# B&R Automation Studio project CControl_Gschneitner (part 18)

```automation-basic
		ENDACTION

	ENDCASE

	InitOK = 1

END_PROGRAM
```

#### CSV01_PRGInit.ab
```automation-basic
PROGRAM _INIT

; Diverse INIT :
; ==============
  InitOK = 0
  CSV01.IW.KOPF_WRITE           = 0
  CSV01.IW.DATA_WRITE           = 0
  CSV01.IW.DATA_WRITE_BEREIT    = 0
  CSV01.IW.RPS_SAVE_STEP_Nr     = 0
  CSV01.IW.RPS_CPYDEL_STEP_Nr   = 0
  CSV01.IW.RPS_DirRead_Start_OK = 0

  M_DatObj_ChangDate = DT#1970-01-01-00:00:00

  strcpy(adr(CSV01.IW.PC_Device), "PC_HD_D")		; PC: Speicherdevice
  strcpy(adr(DatObjInfo_01_Name), "CSV01_CFG")

  CR = $0D			; CR (Enter)
  LF = $0A			; LF (Linefeed)
  StrCRLF[0] = CR	; CR+LF
  StrCRLF[1] = LF	; CR+LF
  StrCRLF[2] = 0	; CR+LF
  StrCRLF[3] = 0	; CR+LF

; Task-Zykluszeit auslesen:
; =========================
  RTInfo(1, RT_Status, ZyklTime, init_reason, task_class)
  ZyklTime = ZyklTime/1000  ; [msek]

END_PROGRAM
```

#### CSV01_PRG.var
```iecst
VAR
	CR : USINT;
	CSV_DatObj1 : CSV_DatObj1_typ;
	CSV_DatObj2 : CSV_DatObj2_typ;
	data_len : UDINT;
	data_len2 : UDINT;
	data_typ : UDINT;
	Datei_Ende : ARRAY[0..1] OF USINT;
	Datensatz : ARRAY[0..60000] OF USINT;
	DatObj_Offset : UDINT;
	DatObj1_Size : UDINT;
	DatObj2_Size : UDINT;
	DatObjInfo_01 : DatObjInfo;
	DatObjInfo_01_Name : ARRAY[0..15] OF USINT;
	DevLink_0 : DevLink;
	DevMemInfo_0 : DevMemInfo;
	dimension : UINT;
	DirCopy_0 : DirCopy;
	DirCreate_0 : DirCreate;
	DirDeleteEx_0 : DirDeleteEx;
	DirInfo_0 : DirInfo;
	DirRead_0 : DirRead;
	DirRead_alt_Date : DATE_AND_TIME;
	DirRead_alt_entry : UDINT;
	DirRead_entry : UDINT;
	DirRead_neu_Date : DATE_AND_TIME;
	DirRead_neu_entry : UDINT;
	DirRead_Nr : UDINT;
	ET : UDINT;
	FileClose_0 : FileClose;
	FileCopy_0 : FileCopy;
	FileCreate_0 : FileCreate;
	FileDelete_0 : FileDelete;
	FileIdent : UDINT;
	FileLength : UDINT;
	FileOpen_0 : FileOpen;
	FileRead_0 : FileRead;
	FileWrite_0 : FileWrite;
	i : UINT;
	ii : UINT;
	init_reason : SINT;
	InitOK : BOOL;
	LF : USINT;
	M_date_Fehler : BOOL;
	M_DatObj_ChangDate : DATE_AND_TIME;
	M_Fehler : BOOL;
	M_File_neu : BOOL;
	M_InitOK : BOOL;
	M_MAX_Fehler : BOOL;
	M_MIN_Fehler : BOOL;
	M_Tag_ID : ARRAY[0..9999] OF BOOL;
	M_Tag_MAX : LREAL;
	M_Tag_MIN : LREAL;
	M_timestamp_Fehler : BOOL;
	M_timestamp_QM_Fehler : BOOL;
	M_UDINT_Fehler : BOOL;
	nxt_adr : UDINT;
	Offset_Ende : UDINT;
	P_Fehler : REFERENCE TO BOOL;
	P_Warnung : REFERENCE TO BOOL;
	pv_adr : UDINT;
	RT_Status : UINT;
	RTC_gettime_Status : UINT;
	status_adr : UINT;
	status_ninfo : UINT;
	Str_date : STRING[10];
	Str_ID : ARRAY[0..11] OF USINT;
	Str_Min : ARRAY[0..11] OF USINT;
	Str_Nachkomma : ARRAY[0..11] OF USINT;
	Str_QM_timestamp : STRING[14];
	Str_RPS_File_Name : ARRAY[0..300] OF USINT;
	Str_Sek : ARRAY[0..11] OF USINT;
	Str_Std : ARRAY[0..11] OF USINT;
	Str_Stellen : ARRAY[0..11] OF USINT;
	Str_timestamp : STRING[23];
	Str_Ziel_File_Name : ARRAY[0..300] OF USINT;
	StrCRLF : ARRAY[0..3] OF USINT;
	StrWork : ARRAY[0..30] OF USINT;
	Tag_MAX_Komma : USINT;
	Tag_MAX_Nachkomma : USINT;
	Tag_MAX_Stellen : USINT;
	Tag_MIN_Komma : USINT;
	Tag_MIN_Nachkomma : USINT;
	Tag_MIN_Stellen : USINT;
	Tag_Nachkomma : USINT;
	task_class : SINT;
	Wert_BOOL : REFERENCE TO BOOL;
	Wert_DINT : DINT;
	Wert_INT : INT;
	Wert_REAL : REAL;
	Wert_SINT : SINT;
	Wert_STRING : ARRAY[0..24] OF USINT;
	Wert_UDINT : UDINT;
	Wert_UINT : UINT;
	Wert_USINT : USINT;
	Zeile_Fertig : BOOL;
	ZyklTime : UDINT;
END_VAR
```

### Data object Logical/CSV/CSV01_CFG (Simple, version 1.00.0) - Tag Configuration

#### CSV01_CFG.dat
```
; ============================================================================================
; ACHTUNG: !!! In diesem Datenmodul dürfen absolut keine Tabulator-Sprünge enthalten sein !!!!
; ============================================================================================

;[ABSCHNITT_CONFIG]
;******************

;<----------------->   -> Länge der 8 nachstehenden Eingabefelder
"1.0.0.1            "  ; USINT[0..19] CSV-Version für Auswertung in Reporting-Software                  z.B.: "1.0.0.1            "
"LATronicCControl   "  ; USINT[0..19] Anlagenname                                                       z.B.: "Heizung_01         "
"CF                 "  ; USINT[0..19]          RPS-Ebene: File-Devicename (CPU Eigenschaften)           z.B.: "CF                 "
"CSV                "  ; USINT[0..19]          RPS-Ebene: Zielordner (nur eine Hirachieebene möglich)   z.B.: "CSV                "
"usb_device         "  ; USINT[0..19] [OPTION] EXTERN   : File-Devicename (CPU Eigenschaften)           z.B.: "USB                "
"CSV                "  ; USINT[0..19] [OPTION] EXTERN   : Zielordner (nur eine Hirachieebene möglich)   z.B.: "CSV                "
"192.168.203.202    "  ; USINT[0..19] [OPTION] PC-Ebene : IP-Adresse PC                                 z.B.: "192.168.203.204    "
"PC_D               "  ; USINT[0..19] [OPTION] PC-Ebene : Windows-Freigabename des Laufwerks am PC  	z.B.: "PC_D               "
"guest              "  ; USINT[0..19] [OPTION] PC-Ebene : Windows-Username (nicht akt. Anmeldung verw.) z.B.: "guest              "
"guest              "  ; USINT[0..19] [OPTION] PC-Ebene : Windows-Userpassword                      	z.B.: "guest              "
"/Daten/Excel/CSV                                                                                   " ;USINT[0..99] [OPTION] PC-Ebene: Zielordner (muß am PC manuell angelegt werden
;<------------------------------------------------------------------------------------------------->

;[ABSCHNITT_DATEN]
;*****************

;TAG-ID          TAG-Variablenname (RPS-Name)                                  TAG-Bezeichung                                   TAG-Einheit                  TAG-MIN           TAG-MAX
;[DINT]                USINT[0..47]                                             USINT[0..59]                                    USINT[0..31]                USINT[0..15]      USINT[0..15]
; 0..9999
;(mit "0"          (RPS-Variablenname)                                          (freier Text)                                   (freier Text)               (Komma=".")       (Komma=".")
;auffüllen!)                                                                                                                                               (=Trend SkalaU)    (=Trend SkalaO)
;                                                                                                                                                          (=Def. Kommast.)  (=Def. Kommast.)
;---->  <--------------------------------------------->   <--------------------------------------------------------->   <----------------------------->   <------------->   <------------->
000001,"gStatusAnlage.Betrieb                          ","ALLG: Betrieb Anlage                                       ","0/1                            ","              0","              1"
000002,"gAktuellesPasswort                             ","ALLG: Aktuelles Passwort                                   ","Num                            ","              0","         999999"
000003,"gStatusAnlage.FrischluftbetriebAktiv           ","ALLG: Frischluftbetrieb Aktiv                              ","0/1                            ","              0","              1"
000004,"gStatusAnlage.UmluftbetriebAktiv               ","ALLG: Umluftbetrieb Aktiv                                  ","0/1                            ","              0","              1"
000005,"gStatusAnlage.Fehler.FehlerNr                  ","ALLG: Fehlernummer                                         ","0-39                           ","              0","             39"
000006,"gStatusAnlage.Fehler.WarnungNr                 ","ALLG: Warnungsnummer                                       ","0-29                           ","              0","             29"
000007,"Aktoren.KompressorModul1.curStep               ","ALLG: Aktueller Schritt Kompressor 1                       ","0-6                            ","              0","              6"
000008,"Aktoren.KompressorModul2.curStep               ","ALLG: Aktueller Schritt Kompressor 2                       ","0-6                            ","              0","              6"
000009,"aiNiederdruckModul1                            ","AI: Niederdruck Modul 1                                    ","bar                            ","            0.0","           30.0"
000010,"aiHochdruckModul1                              ","AI: Hochdruck Modul 1                                      ","bar                            ","            0.0","           30.0"
000011,"aiNiederdruckModul2                            ","AI: Niederdruck Modul 2                                    ","bar                            ","            0.0","           30.0"
000012,"aiHochdruckModul2                              ","AI: Hochdruck Modul 2                                      ","bar                            ","            0.0","           30.0"
000013,"aiFrischluftTemperatur                         ","AI: Frischluft Temperatur                                  ","°C                             ","          -30.0","           70.0"
000014,"aiFrischluftFeuchte                            ","AI: Frischluft rel. Feuchte                                ","%                              ","            0.0","          100.0"
000015,"aiDachluftTemperatur                           ","AI: Dachluft Temperatur                                    ","°C                             ","          -30.0","           70.0"
000016,"aiDachluftFeuchte                              ","AI: Dachluft rel. Feuchte                                  ","%                              ","            0.0","          100.0"
000017,"aiTrockenluftTemperatur                        ","AI: Trockenluft Temperatur                                 ","°C                             ","          -30.0","           70.0"
000018,"aiTrockenluftFeuchte                           ","AI: Trockenluft rel. Feuchte                               ","%                              ","            0.0","          100.0"
000019,"aiAbluftTemperatur                             ","AI: Abluft Temperatur                                      ","°C                             ","          -30.0","           70.0"
000020,"aiAbluftFeuchte                                ","AI: Abluft rel. Feuchte                                    ","%                              ","            0.0","          100.0"
000021,"aiLuftgeschwindigkeit                          ","AI: Luftgeschwindikeit                                     ","m/s                            ","            0.0","           20.0"
000022,"aiDifferenzdruck                               ","AI: Kanaldruck                                             ","Pa                             ","            0.0","         5000.0"
000023,"aiEintrittTemperatur                           ","AI: Eintritt Temperatur                                    ","°C                             ","          -30.0","           70.0"
000024,"aiEintrittFeuchte                              ","AI: Eintritt rel. Feuchte                                  ","%                              ","            0.0","          100.0"
000025,"aiAustrittTemperatur                           ","AI: Austritt Temperatur                                    ","°C                             ","          -30.0","           70.0"
000026,"aiAustrittFeuchte                              ","AI: Austritt rel. Feuchte                                  ","%                              ","            0.0","          100.0"
000027,"aoDrehzahlvorgVentilator1                      ","AO: Drehzahlvorgabe Ventilator 1                           ","%                              ","            0.0","          100.0"
000028,"aoDrehzahlvorgVentilator2                      ","AO: Drehzahlvorgabe Ventilator 2                           ","%                              ","            0.0","          100.0"
000029,"aoDrehzahlvorgKompressorModul1                 ","AO: Drehzahlvorgabe Kompressor Modul 1                     ","%                              ","            0.0","          100.0"
000030,"aoDrehzahlvorgKompressorModul2                 ","AO: Drehzahlvorgabe Kompressor Modul 2                     ","%                              ","            0.0","          100.0"
000031,"aoLeistungsvorgHeizregister                    ","AO: Drehzahlvorgabe Heizregister                           ","%                              ","            0.0","          100.0"
000032,"aoTemperaturvorgWarmluftofen                   ","AO: Temperaturvorgabe Warmluftofen                         ","°C                             ","            0.0","          100.0"
000033,"aoDrehzahlvorgAbluftventilator                 ","AO: Drehzahlvorgabe Abluftventilator                       ","%                              ","            0.0","          100.0"
000034,"gMindestlaufzOelsumpfOk                        ","ALLG: Laufzeit Oelsumpfheizung OK                          ","0/1                            ","              0","              1"
000035,"gStatusAnlage.LuftmengeAktuell                 ","ALLG: Luftmenge Aktuell                                    ","m³/h                           ","            0.0","      9999999.9"
000036,"di24VDCinternIstOk                             ","Status DI Absicherung 24VDC                                ","0/1                            ","              0","              1"
000037,"diNiederdruckOkModul1                          ","Status DI Niederdruck OK Modul 1                           ","0/1                            ","              0","              1"
000038,"diHochdruckOkModul1                            ","Status DI Hochdruck OK Modul 1                             ","0/1                            ","              0","              1"
000039,"diNiederdruckOkModul2                          ","Status DI Niederdruck OK Modul 2                           ","0/1                            ","              0","              1"
000040,"diHochdruckOkModul2                            ","Status DI Hochdruck OK Modul 2                             ","0/1                            ","              0","              1"
000041,"diKopftempKompressorModul1                     ","Status DI Kopftemperatur Kompressor Modul 1                ","0/1                            ","              0","              1"
000042,"diKopftempKompressorModul2                     ","Status DI Kopftemperatur Kompressor Modul 2                ","0/1                            ","              0","              1"
000043,"diOeldruckKompressorModul1                     ","Status DI Öldruck Kompressor Modul 1                       ","0/1                            ","              0","              1"
000044,"diOeldruckKompressorModul2                     ","Status DI Öldruck Kompressor Modul 2                       ","0/1                            ","              0","              1"
000045,"diVollschutzKompressorModul1                   ","Status DI Vollschutz Kompressor Modul 1                    ","0/1                            ","              0","              1"
000046,"diVollschutzKompressorModul2                   ","Status DI Vollschutz Kompressor Modul 2                    ","0/1                            ","              0","              1"
000047,"diBetriebsmldgKompressorModul1                 ","Status DI Betriebsmeldung FU Kompressor Modul 1            ","0/1                            ","              0","              1"
000048,"diBetriebsmldgKompressorModul2                 ","Status DI Betriebsmeldung FU Kompressor Modul 2            ","0/1                            ","              0","              1"
000049,"diAnfEntfeuchterExtern                         ","Status DI Anforderung Entfeuchter Extern                   ","0/1                            ","              0","              1"
000050,"diLeistungsvorgKompressorExtMod1               ","Status DI Leistungsvorgabe Extern Modul 1                  ","0/1                            ","              0","              1"
000051,"diVentilator1InBetrieb                         ","Status DI Betriebsmeldung Ventilator 1                     ","0/1                            ","              0","              1"
000052,"diVentilator2InBetrieb                         ","Status DI Betriebsmeldung Ventilator 2                     ","0/1                            ","              0","              1"
000053,"diDrehzahlbegrVentilator1                      ","Status DI Drehzahlbegrenzung Ventilator 1                  ","0/1                            ","              0","              1"
000054,"diDrehzahlbegrVentilator2                      ","Status DI Drehzahlbegrenzung Ventilator 2                  ","0/1                            ","              0","              1"
000055,"diScheitholzofenInBetrieb                      ","Status DI Betriebsmeldung Scheitholzofen                   ","0/1                            ","              0","              1"
000056,"diWarmluftofenInBetrieb                        ","Status DI Betriebsmeldung Warmluftofen                     ","0/1                            ","              0","              1"
000057,"diNotstromaggregatInBetrieb                    ","Status DI Betriebsmeldung Notstromaggregat                 ","0/1                            ","              0","              1"
000058,"diBox1Offen                                    ","Status DI Klappe Box 1 Offen                               ","0/1                            ","              0","              1"
000059,"diBox1Geschl                                   ","Status DI Klappe Box 1 Geschlossen                         ","0/1                            ","              0","              1"
000060,"diBox2Offen                                    ","Status DI Klappe Box 2 Offen                               ","0/1                            ","              0","              1"
000061,"diBox2Geschl                                   ","Status DI Klappe Box 2 Geschlossen                         ","0/1                            ","              0","              1"
000062,"diBox3Offen                                    ","Status DI Klappe Box 3 Offen                               ","0/1                            ","              0","              1"
000063,"diBox3Geschl                                   ","Status DI Klappe Box 3 Geschlossen                         ","0/1                            ","              0","              1"
000064,"diBox4Offen                                    ","Status DI Klappe Box 4 Offen                               ","0/1                            ","              0","              1"
000065,"diBox4Geschl                                   ","Status DI Klappe Box 4 Geschlossen                         ","0/1                            ","              0","              1"
000066,"diBox5Offen                                    ","Status DI Klappe Box 5 Offen                               ","0/1                            ","              0","              1"
000067,"diBox5Geschl                                   ","Status DI Klappe Box 5 Geschlossen                         ","0/1                            ","              0","              1"
000068,"diBox6Offen                                    ","Status DI Klappe Box 6 Offen                               ","0/1                            ","              0","              1"
000069,"diBox6Geschl                                   ","Status DI Klappe Box 6 Geschlossen                         ","0/1                            ","              0","              1"
000070,"diBypassklappeOffen                            ","Status DI Bypassklappe Offen                               ","0/1                            ","              0","              1"
000071,"diBypassklappeGeschl                           ","Status DI Bypassklappe Geschlossen                         ","0/1                            ","              0","              1"
000072,"diUmschaltklappe1Offen                         ","Status DI Umschaltklappe 1 Offen                           ","0/1                            ","              0","              1"
000073,"diUmschaltklappe2Offen                         ","Status DI Umschaltklappe 2 Offen                           ","0/1                            ","              0","              1"
000074,"diUmschaltklappe1Geschl                        ","Status DI Umschaltklappe 1 Geschlossen                     ","0/1                            ","              0","              1"
000075,"diUmschaltklappe2Geschl                        ","Status DI Umschaltklappe 2 Geschlossen                     ","0/1                            ","              0","              1"
000076,"diAbluftklappeOffen                            ","Status DI Abluftklappe Offen                               ","0/1                            ","              0","              1"
000077,"diAbluftklappeGeschl                           ","Status DI Abluftklappe Geschlossen                         ","0/1                            ","              0","              1"
000078,"diAbluftventInBetrieb                          ","Status DI Abluftventilator in Betrieb                      ","0/1                            ","              0","              1"
000079,"doTrocknungInBetrieb                           ","Status DO Trocknung in Betrieb                             ","0/1                            ","              0","              1"
000080,"doTrocknungStoerung                            ","Status DO Trocknung Störung                                ","0/1                            ","              0","              1"
000081,"doWarmluftofenEin                              ","Status DO Freigabe Warmluftofen                            ","0/1                            ","              0","              1"
000082,"doHeizregisterEin                              ","Status DO Freigabe Heizregister                            ","0/1                            ","              0","              1"
000083,"doKompressorEinModul1                          ","Status DO Freigabe Kompressor Modul 1                      ","0/1                            ","              0","              1"
000084,"doKompressorEinModul2                          ","Status DO Freigabe Kompressor Modul 2                      ","0/1                            ","              0","              1"
000085,"doMagnetventilEinModul1                        ","Status DO Magnetventil Modul 1                             ","0/1                            ","              0","              1"
000086,"doMagnetventilEinModul2                        ","Status DO Freigabe Magnetventil Modul 2                    ","0/1                            ","              0","              1"
000087,"doOelsumpfheizungEinModul1                     ","Status DO Ölsumpfheizung Modul 1                           ","0/1                            ","              0","              1"
000088,"doOelsumpfheizungEinModul2                     ","Status DO Freigabe Ölsumpfheizung Modul 2                  ","0/1                            ","              0","              1"
000089,"doVentilator1Ein                               ","Status DO Freigabe Ventilator 1                            ","0/1                            ","              0","              1"
000090,"doVentilator2Ein                               ","Status DO Freigabe Ventilator 2                            ","0/1                            ","              0","              1"
000091,"doNotstromaggregatEin                          ","Status DO Freigabe Notstromaggregat                        ","0/1                            ","              0","              1"
000092,"doBypassklappeOeffnen                          ","Status DO Bypassklappe Freigabe                            ","0/1                            ","              0","              1"
000093,"doAbluftklappeFreigabe                         ","Status DO Abluftklappe Freigabe                            ","0/1                            ","              0","              1"
000094,"doAbluftventilatorEin                          ","Status DO Freigabe Abluftventilator                        ","0/1                            ","              0","              1"
000095,"doUmluftklappe1Freigabe                        ","Status DO Umluftklappe 1 Freigabe                          ","0/1                            ","              0","              1"
000096,"doUmluftklappe2Freigabe                        ","Status DO Umluftklappe 2 Freigabe                          ","0/1                            ","              0","              1"
000097,"doFreigabeBox1                                 ","Status DO Boxenklappe 1 Öffnen                             ","0/1                            ","              0","              1"
000098,"doFreigabeBox2                                 ","Status DO Boxenklappe 2 Öffnen                             ","0/1                            ","              0","              1"
000099,"doFreigabeBox3                                 ","Status DO Boxenklappe 3 Öffnen                             ","0/1                            ","              0","              1"
000100,"doFreigabeBox4                                 ","Status DO Boxenklappe 4 Öffnen                             ","0/1                            ","              0","              1"
000101,"doFreigabeBox5                                 ","Status DO Boxenklappe 5 Öffnen                             ","0/1                            ","              0","              1"
000102,"doFreigabeBox6                                 ","Status DO Boxenklappe 6 Öffnen                             ","0/1                            ","              0","              1"
000103,"doBrandschutzklappeAuf                         ","Status DO Brandschutzklappe Öffnen                         ","0/1                            ","              0","              1"
000104,"doAbluftklappeFreigabe                         ","Status DO Abluftklappe Öffnen                              ","0/1                            ","              0","              1"
000105,"doAbluftventilatorEin                          ","Status DO Abluftventilator Ein                             ","0/1                            ","              0","              1"
000106,"Nutzungsdaten.BstGes.Kompressor1Std            ","Betriebsstunden Gesamt: Kompressor 1                       ","h                              ","              0","        9999999"
000107,"Nutzungsdaten.BstGes.Kompressor2Std            ","Betriebsstunden Gesamt: Kompressor 2                       ","h                              ","              0","        9999999"
000108,"Nutzungsdaten.BstGes.Ventilator1Std            ","Betriebsstunden Gesamt: Ventilator 1                       ","h                              ","              0","        9999999"
000109,"Nutzungsdaten.BstGes.Ventilator2Std            ","Betriebsstunden Gesamt: Ventilator 2                       ","h                              ","              0","        9999999"
000110,"Nutzungsdaten.BstGes.WarmluftofenStd           ","Betriebsstunden Gesamt: Warmluftofen                       ","h                              ","              0","        9999999"
000111,"Nutzungsdaten.BstGes.HeizregisterStd           ","Betriebsstunden Gesamt: Heizregister                       ","h                              ","              0","        9999999"
000112,"Nutzungsdaten.BstGes.Box1Std                   ","Betriebsstunden Gesamt: Box 1                              ","h                              ","              0","        9999999"
000113,"Nutzungsdaten.BstGes.Box2Std                   ","Betriebsstunden Gesamt: Box 2                              ","h                              ","              0","        9999999"
000114,"Nutzungsdaten.BstGes.Box3Std                   ","Betriebsstunden Gesamt: Box 3                              ","h                              ","              0","        9999999"
000115,"Nutzungsdaten.BstGes.Box4Std                   ","Betriebsstunden Gesamt: Box 4                              ","h                              ","              0","        9999999"
000116,"Nutzungsdaten.BstGes.Box5Std                   ","Betriebsstunden Gesamt: Box 5                              ","h                              ","              0","        9999999"
000117,"Nutzungsdaten.BstGes.Box6Std                   ","Betriebsstunden Gesamt: Box 6                              ","h                              ","              0","        9999999"
000118,"Nutzungsdaten.BstGes.OelsumpfheizungStd        ","Betriebsstunden Gesamt: Oelsumpfheizung                    ","h                              ","              0","        9999999"
000119,"Nutzungsdaten.BstGes.Abtauung1Std              ","Betriebsstunden Gesamt: Abtauung Modul 1                   ","h                              ","              0","        9999999"
000120,"Nutzungsdaten.BstGes.Abtauung2Std              ","Betriebsstunden Gesamt: Abtauung Modul 2                   ","h                              ","              0","        9999999"
000121,"Nutzungsdaten.BstGes.AbluftventStd             ","Betriebsstunden Gesamt: Abluftventilator                   ","h                              ","              0","        9999999"
000122,"Nutzungsdaten.BstGes.FrischluftbetrStd         ","Betriebsstunden Gesamt: Frischluftbetrieb                  ","h                              ","              0","        9999999"
000123,"Nutzungsdaten.BstGes.UmluftbetrStd             ","Betriebsstunden Gesamt: Umluftbetrieb                      ","h                              ","              0","        9999999"
000124,"Nutzungsdaten.Energiemessung.LeistungAktuell   ","Energiemessung: Leistung Aktuell                           ","kW                             ","            0.0","        99999.9"
000125,"Nutzungsdaten.Energiemessung.EnergieTag        ","Energiemessung: Energie Tag                                ","kWh                            ","            0.0","      9999999.9"
000126,"Nutzungsdaten.Energiemessung.EnergieGesamt     ","Energiemessung: Energie Gesamt                             ","kWh                            ","            0.0","      9999999.9"
000127,"gStatusAnlage.WetterIstSchlecht                ","ALLG: Wetter ist schlecht                                  ","0/1                            ","              0","              1"
000128,"doEntfFremdFreigabe                            ","Status DO Freigabe Entfeuchter Fremdgerät                  ","0/1                            ","              0","              1"
000129,"diEntfeuchterFremdInBetrieb                    ","Status DI Betriebsmldg Entfeuchter Fremdgerät              ","0/1                            ","              0","              1"
000130,"diEntfeuchterFremdStoerung                     ","Status DI Störmeldung Entfeuchter Fremdgerät               ","0/1                            ","              0","              1"
000131,"diHeizregisterFrostschutz                      ","Thermostateingang Frostschutz Heizregister	             ","0/1                            ","              0","              1"
```

### Program Logical/Sitemanager/Sitemanager (IEC) - AsTCP Client Application

#### Client.st - Cyclic code
```iecst
(********************************************************************
* EMAIL Client für Sitemanager
*
* AUTH: ErKai KATOMA 20210516
*********************************************************************)

PROGRAM _CYCLIC

	//Betriebsparameter übergeben
	loc_EMailAlarmierungEin := Betriebsparameter.Fernalarmierung.EMailAlarmierungEin;
	EMail[0] := Betriebsparameter.Fernalarmierung.MailAdresse[0];
	EMail[1] := Betriebsparameter.Fernalarmierung.MailAdresse[1];
	EMail[2] := Betriebsparameter.Fernalarmierung.MailAdresse[2];
	EMail[3] := Betriebsparameter.Fernalarmierung.MailAdresse[3];

	//1. Alarm aus Visu auslesen
	//**************************
	IF VC_HANDLE = 0 THEN
		VC_HANDLE := VA_Setup(1, 'Visu');
	END_IF

	IF hmiButtons.QuitFehler THEN
		loc_FehlerAusgelesen	:= FALSE;
	END_IF

	IF gStatusAnlage.Fehler.SummeFehler AND NOT loc_FehlerAusgelesen AND loc_EMailAlarmierungEin THEN
		Access_Status := VA_Saccess(1, VC_HANDLE);
		IF Access_Status = 0 THEN
			AlarmLen 			:= 80;
			cSeparator 			:= 45; //Bindestrich
			uiAlarmType 		:= 1; //Ersten Alarm auslesen
			cDateTimeFormat 	:= 6; //Kein Datum, keine Uhrzeit

			GetActAlarmList_Status := VA_GetActAlarmList(1, VC_HANDLE, (ADR(AlarmString)), (ADR(AlarmLen)), uiAlarmType, cSeparator, cDateTimeFormat);

			IF GetActAlarmList_Status = 0 THEN
				loc_FehlerAusgelesen	:= TRUE;
				EMailText				:= AlarmString;
				Send					:= TRUE;
			END_IF
			VA_Srelease(1, VC_HANDLE);
		END_IF
	END_IF

	IP_ADRESS := ADR(Betriebsparameter.Allgemein.DefaultGateway);
	//IP_ADRESS := ADR('10.0.0.1');
	IP_PORT := 26864;

	Sendstring:=SLASH;
	UseComma:=FALSE;
	CommaString:='';

	IF EMail[0] <> '' THEN
		resultString:= CONCAT(LEFTBRACKET, EMail[0]);
		IF EMail[1]='' AND EMail[2]='' AND EMail[3]='' THEN
			resultString:= CONCAT(resultString, RIGHTBRACKET);
		END_IF;

		Sendstring:= CONCAT(Sendstring, resultString);
		UseComma:=TRUE;
	END_IF;

	IF EMail[1] <> '' THEN
		IF UseComma THEN
			CommaString:=COMMA;
			resultString:= COMMA;
		END_IF;
		resultString:= CONCAT(resultString, EMail[1]);
		IF EMail[2]='' AND EMail[3]='' THEN
			resultString:= CONCAT(resultString, RIGHTBRACKET);
		END_IF;

		Sendstring:= CONCAT(Sendstring,resultString);
		UseComma:=TRUE;
	END_IF;

	IF EMail[2] <> '' THEN
		IF UseComma THEN
			CommaString:=COMMA;
			resultString:= COMMA;
		END_IF;
		resultString:= CONCAT(resultString, EMail[2]);
		IF EMail[3]='' THEN
			resultString:= CONCAT(resultString, RIGHTBRACKET);
		END_IF;

		Sendstring:= CONCAT(Sendstring,resultString);
		UseComma:=TRUE;
	END_IF;

	IF EMail[3] <> '' THEN
		IF UseComma THEN
			CommaString:=COMMA;
			resultString:= COMMA;
		END_IF;
		resultString:= CONCAT(resultString, EMail[3]);
		resultString:= CONCAT(resultString, RIGHTBRACKET);
		Sendstring:= CONCAT(Sendstring,resultString);
		UseComma:=TRUE;
	END_IF;

	Sendstring:= CONCAT(Sendstring,SLASH);

	Sendstring:= CONCAT(Sendstring,EMailText);

	CASE Client.sStep OF

		0:	IF Send THEN
				ErrNr:=0;
				ErrorText:='';
				Client.sStep := 1;
			END_IF;

		(*Open*)
		 1: Client.TcpOpen_0.enable := 1;
			Client.TcpOpen_0.pIfAddr := 0;
			Client.TcpOpen_0.port := 26864;
			Client.TcpOpen_0.options := 0;
			Client.TcpOpen_0;

			IF Client.TcpOpen_0.status = 0 THEN
				Client.sStep := 5;
			ELSIF Client.TcpOpen_0.status = ERR_FUB_BUSY THEN
			  (*nicht feritg*)
			ELSE
				ErrNr:= Client.TcpOpen_0.status;
				Client.sStep := 100;
			END_IF

			(*Set Linger*)
		 5: Client.linger_opt.lLinger := 0;
			Client.linger_opt.lOnOff := 1;

		 	Client.TcpIoctl_0.enable := 1;
			Client.TcpIoctl_0.ident := Client.TcpOpen_0.ident;
			Client.TcpIoctl_0.ioctl := tcpSO_LINGER_SET;
			Client.TcpIoctl_0.pData := ADR(Client.linger_opt);
			Client.TcpIoctl_0.datalen := SIZEOF(Client.linger_opt);
   			Client.TcpIoctl_0;

			IF Client.TcpIoctl_0.status = 0 THEN
				Client.sStep := 10;
			ELSIF Client.TcpIoctl_0.status = ERR_FUB_BUSY THEN
			  (* hmhm.... *)
			ELSE
				ErrNr:= Client.TcpIoctl_0.status;
				Client.sStep := 100;
			END_IF

		10: (* Connect*)
			Client.TcpClient_0.enable := 1;
			Client.TcpClient_0.ident := Client.TcpOpen_0.ident;
			Client.TcpClient_0.portserv := IP_PORT;
			Client.TcpClient_0.pServer := IP_ADRESS;
			Client.TcpClient_0;

			IF Client.TcpClient_0.status = 0 THEN
				Client.sStep := 20;
			ELSIF Client.TcpClient_0.status = ERR_FUB_BUSY THEN
			  (* dudu.... *)
			ELSIF Client.TcpClient_0.status = tcpERR_INVALID THEN
				ErrNr:= Client.TcpClient_0.status;
				ErrorText:= 'ERR_INVALID, Fehler Verbindungsaufbau';
				Client.sStep := 40;
			ELSE
				ErrNr:= Client.TcpClient_0.status;
				Client.sStep := 100;
			END_IF

		20: (* Send*)
			Client.TcpSend_0.enable := 1;
			Client.TcpSend_0.ident := Client.TcpOpen_0.ident;
			Client.TcpSend_0.pData := ADR(Sendstring);
			Client.TcpSend_0.datalen := LEN(Sendstring);
			Client.TcpSend_0.flags := 0;
			Client.TcpSend_0;

			IF Client.TcpSend_0.status = 0 THEN
				Client.sStep := 40;
			ELSIF Client.TcpSend_0.status = ERR_FUB_BUSY THEN
			  (* lala..... *)
			ELSIF (Client.TcpSend_0.status = tcpERR_SENTLEN) OR (Client.TcpSend_0.status = tcpERR_NOT_CONNECTED) THEN
				CASE Client.TcpSend_0.status OF
					tcpERR_SENTLEN: ErrorText:= 'ERR_SENTLEN Die, übernommene Datenlänge entspricht nicht der angegebenen Datenlänge.';
					tcpERR_NOT_CONNECTED: ErrorText:= 'ERR_NOT_CONNECTED, Die Verbindung wurde beendet (Gegenstelle).';
				END_CASE
				ErrNr:= Client.TcpSend_0.status;
				Client.sStep := 40;
			ELSE
				ErrNr:= Client.TcpSend_0.status;
				Client.sStep := 100;
			END_IF

		40: (* Close *)
			Client.TcpClose_0.enable := 1;
			Client.TcpClose_0.ident := Client.TcpOpen_0.ident;
			Client.TcpClose_0.how := 0;
			Client.TcpClose_0;

			IF Client.TcpClose_0.status = 0 THEN
				Client.sStep := 0;
				Send:=FALSE;
			ELSIF Client.TcpClose_0.status = ERR_FUB_BUSY THEN
				(*tütü... *)
			ELSE
				ErrNr:= Client.TcpClose_0.status;
				Client.sStep := 100;
			END_IF

		(*Error*)
		100:
			CASE ErrNr OF
				32600: ErrorText:= 'ERR_INVALID_IDENT Der angegebene Ident ist nicht zulässig.';
				32601: ErrorText:= 'ERR_NOMORE_IDENTS, Es konnte kein weiterer Ident reserviert werden.';
				32602: ErrorText:= 'ERR_ALREADY_EXIST, Es existiert bereits ein Socket, der auf diese Portnummer';
				32603: ErrorText:= 'ERR_PARAMETER, Ungültige Parameter.';
				32604: ErrorText:= 'ERR_INVALID_IOCTL, Ungültiges IO-Control.';
				32606: ErrorText:= 'ERR_SENTLEN Die, übernommene Datenlänge entspricht nicht der angegebenen Datenlänge.';
				32607: ErrorText:= 'ERR_WOULDBLOCK, Daten konnten nicht in den Sendepuffer des Sockets übernommen werden.';
				32608: ErrorText:= 'ERR_INVALID, Fehler Verbindungsaufbau';
				32609: ErrorText:= 'ERR_NOT_CONNECTED, Die Verbindung wurde beendet (Gegenstelle).';
				32650: ErrorText:= 'ERR_SOCKET_CREATE, Ressourcenproblem im System. Es konnte kein Socket mehr angelegt werden.';
				32651: ErrorText:= 'ERR_SOCKET_BIND, Problem beim Binden an die Portnummer bzw. an die ermittelte Ip-Adresse';
				32612: ErrorText:= 'ERR_INTERFACE, Die angegebene Interface-Adresse ist ungültig.';
				32699: ErrorText:= 'ERR_SYSTEM, Interner Fehler beim Senden.';
				65534: ErrorText:= 'ERR_FUB_ENABLE_FALSE, Fub nicht enabled. FUB enablen.';
				65535: ErrorText:= 'ERR_FUB_BUSY, Fub arbeitet noch.';
			END_CASE
			Send:=FALSE;
			Client.sStep:=0;
	END_CASE

END_PROGRAM
```

#### Client.typ - TCP Client Variables
```iecst
TYPE
	Client_typ : 	STRUCT
		sStep : UINT;
		TcpOpen_0 : TcpOpen;
		TcpClient_0 : TcpClient;
		TcpRecv_0 : TcpRecv;
		TcpSend_0 : TcpSend;
		TcpIoctl_0 : TcpIoctl;
		TcpClose_0 : TcpClose;
		linger_opt : tcpLINGER_typ;
	END_STRUCT;
END_TYPE
```

#### Client.var - Data for Client Task
```iecst
VAR
	Sendstring : STRING[350] := '';
	Client : Client_typ := (0);
	EMailText : STRING[80] := '';
END_VAR
VAR CONSTANT
	SLASH : STRING[1] := '/';
	LEFTBRACKET : STRING[1] := '<';
	RIGHTBRACKET : STRING[1] := '>';
	COMMA : STRING[1] := ',';
END_VAR
VAR
	EMail : ARRAY[0..3] OF STRING[80] := [4('')];
	UseComma : BOOL := FALSE;
	CommaString : STRING[1] := '';
	Send : BOOL := FALSE;
	resultString : STRING[350] := '';
	ErrorText : STRING[80] := '';
	ErrNr : UINT := 0;
	IP_PORT : UINT := 0;
	IP_ADRESS : UDINT := 0;
END_VAR
(*VC - Variablen ===============================================================================================================================*)
VAR
	VC_HANDLE : UDINT;
	AlarmString : STRING[100];
	AlarmLen : DINT;
	uiAlarmType : UINT;
	cDateTimeFormat : USINT;
	cSeparator : USINT;
	Access_Status : UINT;
	GetActAlarmList_Status : UINT;
	loc_FehlerAusgelesen : BOOL;
	loc_EMailAlarmierungEin : BOOL;
END_VAR
```

### versionsinfo.txt
```
##########################################################
LaTronic CControl 3.07, 4.07 & 4.07 Plus Versionshistorie
##########################################################

--------------------------------------------------------------------------------------------
Version 0.0.0	     	Initialversion			2022.05.19					RL
--------------------------------------------------------------------------------------------

--------------------------------------------------------------------------------------------
Version 0.0.1	     	new/change/fix			2022.06.01					RL
--------------------------------------------------------------------------------------------

Neu:
****
- Optionen fuer Verhalten der Ventilatoren bei Klappenumschaltungen hinzugefuegt (Beide oder nur zustaendigen Ventilator
bei Umschaltungen Boxenklappen, Umluftklappen und Bypassklappe).
- Option "Abluftklappe im Frischluftbetrieb immer offen" hinzugefuegt (Abluftklappe oeffnet im Frischluftbetrieb unabhaengig von der
eingestellten Abluftfeuchte, wenn Klappe auf Automatik gestellt).
- Option "Alle Boxenklappen im Stillstand schliessen" hinzugefuegt.
- Trockengut "Mais" und "Getreide" hinzugefuegt.
- VNC-Viewer bei allen Konfigurationen hinzugefuegt.
- "Notbetrieb" fuer alle Boxen und Ventilatoren hinzugefuegt (fuer Auskuehlphase Warmluftofen). Boxenklappen und Ventilatoren bleiben aktiv,
bis Auskuehlphase abgeschlossen ist.
- Funktion zum Kopieren der XML-Parametersaetze auf einen USB-Stick hinzugefuegt.
- Zusatztexte hinzugefuegt, wenn Trocknungsgeraete wegen Tarifabschaltung aus sind (Vorlaufzeit Tarifabschaltung).
- Zoom fuer Trendkurven hinzugefuegt.
- Hopfen und Kraeuter bei Trockenguetern hinzugefuegt.
- Automatisches Laden der Werksparameter bei neuen Displays hinzugefuegt.
- Franzoesische Sprache hinzugefuegt.
- Energiemessmodul in allen Hardwarekonfigurationen hinzugefuegt.
- Trockengut "Holz" hinzugefuegt (Visualisierung/Visu, hmiMain).
- Modulueberwachungen fuer alle Hardwarekonfigurationen hinzugefuegt (IO/io307, io407, io407Plus).

Aenderungen:
***********
- Wenn Strombegrenzung der Ventilatoren aktiv ist (Zeitfenster oder digitaler Eingang), geht der Luftentfeuchter bei Ueberschreiten
des max. Hochdrucks in den Standby-Betrieb (wie bei Klappenumschaltungen).
- Warnung "Entfeuchter Hochdruck max." wird nur generiert, wenn keine Strombegrenzung oder Klappenumschaltung aktiv ist.
- Nur Option "Abluftklappe" ODER "Abluftventilator" erlauben, beide Optionen sind nicht moeglich.
- Beim Abschalten der Ventilatoren die Freigabe erst wegschalten, wenn Min-Drehzahl erreicht wurde.
- Buttons und Slider fuer Ausstattung und Konfiguration Aktoren Boxen sperren, wenn Benutzerebene < LASCO.
- Beim Wechsel von Betrieb auf AUS einer Box -> Arrays Zeitfenster Intervallbetrieb und Nachtrockung auf 0 setzen.
- Entfeuchter, Warmluftofen und Heizregister erst freigeben, wenn zustaendiger Ventilator in Betrieb ist.
- Boxen koennen auch gestartet werden, wenn Summenfehler aktiv (Sperren Visu entfernt, Wechsel in Betriebsart "BETRIEB" trotz Summenfehler).
- Signal "cmdAnlage.FehlerStopp" entfernt (Trocknung kann trotz Fehler gestartet werden bzw. wird nicht mehr automatisch gestoppt).
- Ansteuerung Bypassklappe geaendert (actionBetrieb).
- Skalierung Drehzahlvorgabe Kompressor Modul 1 und 2: Min auf "0" gesetzt. (IO/io307, io407Plus).
- Drehzahlvorgaben von FU Kompressor angepasst (Libaries/LascoEntfV2/fbEntfKompressor).
- Doppelmodul nur bei bei den Typen 7, 8, 9 und 10 (10 ist Reserve) (IO/aktorenMapping).
- Fehlermeldungen Entfeuchter Temperatur Eintritt Min/Max nur ausgeben, wenn Entfeuchter angefordert. (Alarmsystem/Alarm).
- Drehzahlvorgabe Heizregister auf Min. setzen, wenn Heizregister nicht freigegeben (Regelung/Leistung).
- Ventilatoren: Wenn eingestellte Drehzahl bei Klappenumschaltungen auf MIN (30%) -> Ventilator ausschalten (Libaries/LascoBoxen/fbBoxenVentKlappen).
- Automatikbetrieb von Abluftklappe auch im Stillstand aktivieren (Ablaufsteuerung/actionStillstand).
- Parameter "Hochdruck Max." und "Verzoegerung Standy, wenn Hochdruck Max." bereits ab Benutzerebene "LASCO" einstellbar (Visualisierung/Visu).

Fehlerbehebungen:
*****************
- Indexe fuer Fehler, Systemmeldungen und Warnungen angepasst (fuer Filter bei historischen Alarmen).
- Fehler Laufzeitueberwachungen Boxenklappen nur generieren, wenn Klappe verwendet wird.
- Min/Max Werte bei Eingabefeldern Detailansicht Klappen hinzugefuegt.
- Struktur "hmiAktuell" remanent deklariert, da ansonsten die Betriebsart der Box nach Stromausfall geaendert wird.
- Taste "Datenaufzeichnung auf USB kopieren" zuruecksetzen, wenn Kopiervorgang fertig.
- Diverse CSV-Variablen in Datencontainer aktualisiert.
- 4.07Plus: Signalart Luftgeschwindigkeitssensor auf 0-10V geaendert.
- Restlaufzeit Oelsumpfheizung in hmiParameter speichern (war Betriebsparameter).
- 4.07 Plus: DO Freigabe Ventilator 2 von Ausgang 2 auf 1 geaendert.
- Doppelbelegung von Funktionsbausteinen entfernt (Alarmsystem/Alarm).
- Zusatztext "Auskuehlzeit Scheitholzofen" Fehlerbehebung (Visualisierung/hmiConnect).
- Zusatztext "Warten bis Entfeuchter im Stillstand" auch anzeigen, wenn Boxen pausiert werden (Visualisierung/hmiConnect).
- Status Umluftklappen "Aktiv" nur generieren, wenn Klappe in Ausstattung vorhanden (IO/aktorenMapping).
- Digitale Eingaenge "diOeldruckKompressorModul2" und "diKopftemperaturKompressorModul2" ausgetauscht (IO/io407Plus).
- Eingang "BetriebsmeldungVent" von Kompressor Modul 2 korrigiert (IO/aktorenMapping).
- "StoerungOut" von Funktionsbaustein "fbEntfKompressor" nicht automatisch ruecksetzen, muss manuell quittiert werden (Libaries/LaEntfV2/fbEntfKompressor).
- Digialen Eingang "BetriebsmldgKompressorMod1" im IO-Test korrigiert (IO/io407Plus).
- 3.07: Je nach Ausstattung Analogeingaenge und Statuseingaenge als Dachluft- oder Frischluftsensor skalieren (IO/io307).

--------------------------------------------------------------------------------------------
Version 1.0.0	     	Erstversion Auslieferung		2022.06.22					RL
--------------------------------------------------------------------------------------------

--------------------------------------------------------------------------------------------
Version 1.1.0	     	new/fix/change					2022.09.22					RL
--------------------------------------------------------------------------------------------

Neu:
****
- Slowenische Sprache hinzugefuegt (Visualisierung).
- Laden und Erstellen eines Parametersatzes sperren, wenn Filename "307Werk", "407Werk" oder "407PlusWerk" ist (Visualisierung/Visu).

Aenderungen:
***********
- Die letzten 100 Ereignisse in der Alarmhistorie werden remanent aufgezeichnet (Visualisierung/Visu).

Fehlerbehebungen:
*****************
- Temperatur Austritt Entfeuchter: Falsch angehaengten Wert in Visu korrigiert (Visualisierung/hmiMain).

TODO:
*****
- Verzoegerungszeit Umschaltung Klappen, bis Endlage erreicht wurde?

--------------------------------------------------------------------------------------------
Version 1.1.1	     	fix								2022.09.22					RL
--------------------------------------------------------------------------------------------

Fehlerbehebungen:
*****************
- Bei Anlagen mit Bypassklappe: Freigabe Entfeuchter war von Betrieb des zustaendigen Ventilators abhaengig. Dadurch war die Freigabe des Kompressors immer nur solange
vorhanden, bis die Bypassklappe umgeschaltet wurde (staendiges hin- und herschalten der Klappen). Geaendert, dass die Kompressor-Freigabe erhalten bleibt, wenn die Ventilatoren
kurzzeitig zum Umschalten der Klappen ausgeschaltet werden (Ablaufsteuerung/Ablaufstrg/actionBetrieb).

--------------------------------------------------------------------------------------------
Version 1.1.2	     	new								2023.05.03					RL
--------------------------------------------------------------------------------------------

Neu:
****
- Sensor Kanaldruck fuer Konfiguration 3.07 hinzugefuegt (IO/io307).

--------------------------------------------------------------------------------------------
Version 1.2.0	     	new/change						2023.05.26					RL
--------------------------------------------------------------------------------------------

Neu:
****
- Neue Visualisierung fuer CControl 3.04 hinzugefuegt (PPC30 4 Zoll).
- Hardwarekonfiguration & IO-mapping fuer CControl 3.04 hinzugefuegt.
- Ausgaenge oeffnen/schliessen fuer Klappenansteuerungen (Umluftklappen, Bypassklappe, Abluftklappe, ...) hinzugefuegt.
- Inselbetrieb fuer Luftentfeuchter hinzugefuegt.

Aenderungen:
***********
- Statuseingang "rel. Feuchte MAX" bei allen Feuchte/Temperaturfuehlern fuer Fehlergenerierung entfernt (fuehrt ansonsten zu Fehler, wenn rel. Feuchte tatsaechlich bei 100% ist) (Alarmsystem/Alarm)

--------------------------------------------------------------------------------------------
Version 2.0.0	     	new/change						2024.07.04					RL
--------------------------------------------------------------------------------------------

Neu:
****
- Konfiguration fuer HB4000 & HB3000 hinzugefuegt.
- Betriebsmodus "Dauerbetrieb" in "Automatik" umbenannt. Bei Anlagen ohne Luftaufbereitung (Kaltbelueftungen) wechselt die Box
bei schlechter Witterung in einen Puls/Pausebetrieb (wie bei HB3000/HB4000). Die Bestimmung der Witterungsverhaeltnisse kann fuer jede
Box seperat eingestellt werden.
- Entfeuchter Fremdgeraet hinzugefuegt (Ansteuerung von Frigopol/Baier Luftentfeuchtern).
- Option fuer Stellung Umluftklappen im Stillstand (Frischluft oder Umluft), wenn Umluftklappen im Automatikbetrieb sind.
- Option "Endlagen" fuer alle Klappenantriebe (ausgenommen Abluftklappe) hinzugefuegt. Wird die Option ausgeschaltet (keine Endlagen vorhanden), wird ueber die
eingestellte Laufzeit der Klappe die Fahrt simuliert (Ventilator bleibt fuer die Laufzeit ausgeschaltet/reduziert).

Aenderungen:
***********
- Im Stillstand Umluftklappen & Abluftklappe nicht automatisch umschalten (Ablaufsteuerung, Ablaufstrg/actionBetrieb).
- Default-Gateway als DEV1-Port verwenden (war fix auf 10.0.0.1 eingestellt) (Sitemanager/Sitemanager).
- Parameter "Einschaltverzoegerung Entfeuchter" von 30 auf 120 Sekunden im Standardparametersatz aller Entfeuchtersteuerungen geaendert (lt. Werner).

TODO:
*****
- Uebersetzungen ergaenzen (Aktuell nur Deutsch und Englisch verfuegbar)
- Visu 3.04
- Standardparameter restliche Steuerungen

--------------------------------------------------------------------------------------------
Version 2.1.0	     	new/change						2024.12.02					RL
--------------------------------------------------------------------------------------------

Neu:
****
- Option Stellung Umluftklappen im Stillstand: Stellung kann fuer Klappe 1 und 2 separat eingestellt werden.
- Konfiguration fuer CControl 2.07 hinzugefuegt.

Aenderungen:
***********
- Schlechtwetterbetrieb: Anstatt der Boxenlaufzeit (in Stunden) wird die aktuelle Stufe durch die Trockengutfeuchte (%) bestimmt (manuelle Eingabe durch Bediener).

--------------------------------------------------------------------------------------------
Version 2.1.1	     	new/change						2025.05.07					RIG
--------------------------------------------------------------------------------------------

Aenderungen:
***********
- Bugfix - Bei der Karte X20CM8281f war die Modulueberwachung aktiviert. Dies fuehrte dazu das die Steuerung nicht hochgefahren ist und beim Booten im Servicemodus haengen blieb.

--------------------------------------------------------------------------------------------
Version 2.1.2	     	new/change						2025.05.15					RIG
--------------------------------------------------------------------------------------------

Aenderungen:
***********
- Bugfix - Fehler Betriebsmeldung "Entfeuchter Fremdgeraet" wurde gesetzt obwohl Fremdgeraet nicht aktiviert war

--------------------------------------------------------------------------------------------
Version 2.1.3	     	new/change						2025.06.12					RIG
--------------------------------------------------------------------------------------------

Neu:
****
- Parametersaetze fuer 3.04 und 3.07 erstellt. Wurden aus 4.07 kopiert!
- Registerflache <Property ID="[2]" DataType="REAL" Value="3.3" /> von 3.8 auf 3.3 geaendert. Laut Werner war das schon immer falsch.

Aenderungen:
***********
- Bugfix - Klappenansteuerung Anzugsverzoegerung fuer oeffnen und schliessen der Klappen eingebaut. Dient dazu das andere Relaise abfallen zu lassen bevor das andere geschaltet wird. Verhindert Doppelansteuerung.

--------------------------------------------------------------------------------------------
Version 2.1.4	     	new/change						2025.01.29					RIG
--------------------------------------------------------------------------------------------

Neu:
****
- Frostschutz Heizregister. Bei sehr kalten Temperaturen schaltet ein Thermostat einen Eingang. Ist dieser aktiv wird die
  Kuehlmittelzirkulation aktiviert. Das Heizregister wird so gegen Frostschaeden geschuetzt.

Aenderungen:
***********
- Statuseingang Temperaturwaechter hinzugefuegt. Bei aktivem Eingang ist die Frostschutzlogik aktiv.
- Die Funktion ist nicht ueber die Visu aktivier/deaktivierbar, ist also immer aktiv wenn der Eingang aktiv ist
- Adminkennwort geaendert

--------------------------------------------------------------------------------------------
Version 2.1.5	     	new/change						2026.09.22					RIG
--------------------------------------------------------------------------------------------

Kundenanpassung Gschneitner (CControl 4.07): Die Umluftklappen werden als Warmluft-/Kaltluftumschaltung
verwendet und vom Bediener direkt ueber die Visu geschaltet. Die Anlage kennt nur noch den Frischluftbetrieb.

Neu:
****
- Warmluft-/Kaltluftumschaltung je Ventilator: Die HMI-Buttons in der Klappen-Detailansicht schalten den
  digitalen Ausgang der Umschaltklappe direkt (Klappe angesteuert = Warmluft, stromlos = Kaltluft)
  (Visualisierung/hmiMain, IO/aktorenMapping).
- Statussignale gStatusAnlage.Warmluft1, Warmluft2 und WarmluftAnforderung hinzugefuegt. WarmluftAnforderung
  ist nur gesetzt, wenn mindestens ein laufender Ventilator auf Warmluft steht (Global.typ,
  Ablaufsteuerung/Ablaufstrg/actionUpdateStatus).

Aenderungen:
***********
- Button-Variablen sprechend umbenannt: hmiButtons.changeBetrArtUmluftklappen -> changeWarmluftVent1 und
  hmiButtons.changeBetrArtBypassklappe -> changeWarmluftVent2 (VisuIO.typ, VCShared/DataSources/DataSource.dso,
  Visualisierung/Visu und Visu4Z gDetailsKlappen).
- Betriebsart Umschaltklappen fest auf Frischluft gestellt, die witterungsgefuehrte Umschaltung entfaellt.
  Die Originallogik ist auskommentiert erhalten (Visualisierung/hmiMain, Ablaufsteuerung/Ablaufstrg/actionBetrieb,
  actionStillstand).
- Die Umschaltklappen behalten auch im Stillstand die vom Bediener gewaehlte Stellung
  (Ablaufsteuerung/Ablaufstrg/actionStillstand).
- Heizregister wird abgeschaltet, wenn kein laufender Ventilator auf Warmluft steht: Freigabe und 0-10V Signal
  gehen auf 0 und der PID-Regler wird gesperrt, damit der I-Anteil nicht weiterlaeuft
  (Ablaufsteuerung/Ablaufstrg/actionBetrieb, IO/aktorenMapping, Regelung/Leistung).
- Ventilatorabschaltung waehrend der Umschaltung der Umluftklappen deaktiviert, da die Klappen vom Bediener
  geschaltet werden (IO/aktorenMapping).
- Ventilatorregelung folgt der Warmluft-/Kaltluftumschaltung des jeweiligen Ventilators: Kaltluft verwendet
  die bisherige Frischluftlogik (Fixdrehzahl DrehzahlFixFrischluft), Warmluft die bisherige Umluftlogik
  (Fixdrehzahl DrehzahlFixUmluft oder Luftmengenregelung, je nach Einstellung des Bedieners im
  Ventilator-Popup). Die Variablennamen wurden nicht umbenannt, die Zuordnung ist im Code kommentiert
  (Regelung/Leistung).
- Soll-Luftmenge wird fuer beide Parametersaetze berechnet, da die zwei Ventilatoren unterschiedlich stehen
  koennen und fbBoxenLuftmengen nur eine gemeinsame Betriebsart kennt (Regelung/Leistung).
- Fixdrehzahlvorgabe Ventilator 1 und 2 haengt jetzt an Warmluft1/Warmluft2 statt am anlagenweiten
  Frischluft-/Umluftstatus. Bisher wurde immer DrehzahlFixFrischluft verwendet, der Umluftwert war wirkungslos.
  Gilt fuer alle Zweige: Normalbetrieb, Leistungsreduzierung und Strombegrenzung (Regelung/Leistung).
- Ventilator-Detailansicht umbenannt (nur deutscher Textlayer, Visualisierung/Visu): 'Frischluftbetrieb' ->
  'Kaltluftbetrieb' (TXT_FrischlDachluft) und 'Umluftbetrieb' -> 'Warmluftbetrieb' (gDetailsVentilatoren).
  Anlagenstatus, Betriebsstundenzaehler und Ausstattungsseiten behalten ihre Bezeichnungen.
- Parametersatz 407Werk angepasst: Umschaltklappe 1 und 2 in der Ausstattung aktiviert, Luftmengenregler
  Umluft fuer Ventilator 1 und 2 freigegeben (Kaltluft nur Fixdrehzahl), Betriebsart Umschaltklappen von
  Automatik auf Frischluft (Parametersaetze/407/407Werk.xml).
```
